(* IEC 61131-3 sources: Std_PalletMover/Class/Wewo_LinkedObjectBase, 1 file *)

(* ---- Wewo_LinkedObjectBase.st ---- *)
(*!
<Class
	Name               = "Wewo_LinkedObjectBase"
	Revision           = "0.10"
	RealtimeTask       = "false"
	CyclicTask         = "false"
	BackgroundTask     = "false"
	Sigmatek           = "false"
	OSInterface        = "false"
	HighPriority       = "false"
	Automatic          = "false"
	UpdateMode         = "Prescan"
	SharedCommandTable = "true"
	Objectsize         = "(654,120)"
	Comment            = "Base class for linked objects&#13;&#10;">
	<Channels>
		<Client Name="p_NextObject" Required="false" Internal="false" Comment="Pointer to next object in linked list"/>
		<Client Name="p_PreviousObject" Required="false" Internal="false" Comment="Pointer to previous object in linked list&#13;&#10;(is automatically filled if p_NextObject is connected)"/>
	</Channels>
	<RevDoku>
		<Owner Company="Safan BV" Author="HenOdi"/>
		<Dokumentation Revision="0.10" Date="2012-03-14" Author="HenOdi" Company="Safan BV" Description="Init() Only set p_NextObject durin initCnt=2&#13;&#10;Prepare to remove methodes (add DO_NOT_USE) in future"/>
		<Dokumentation Revision="0.9" Date="2011-11-22" Author="NieTie" Company="Safan BV" Description="Split up Linked List functionality into&#13;&#10;- Linked List Control base&#13;&#10;- Linked List object base&#13;&#10;&#13;&#10;Remove control functionality from "/>
	</RevDoku>
	<Network Name="Wewo_LinkedObjectBase">
		<!-- List of Components in this network -->
		<Components>
			<Object
				Name       = "_base"
				Class      = "WewoBase"
				Position   = "(218,120)"
				Visualized = "false">
				<Channels>
					<Server Name="m_Id"/>
					<Server Name="m_p_Name"/>
					<Server Name="o_ErrorWarningStatus"/>
					<Server Name="ObjectStatus"/>
					<Server Name="ToObject"/>
					<Client Name="c_Group"/>
					<Client Name="op_LogData"/>
					<Client Name="toOsLibTaskObjControl"/>
				</Channels>
			</Object>
		</Components>
		<Comments>
		</Comments>
		<!-- List of Connections in this network -->
		<Connections>
			<Connection Source="this.ToObject" Destination="_base.ToObject" Vertices="(856,210),(684,210),"/>
			<Connection Source="this.ObjectStatus" Destination="_base.ObjectStatus" Vertices="(856,270),(684,270),"/>
			<Connection Source="this.o_ErrorWarningStatus" Destination="_base.o_ErrorWarningStatus" Vertices="(856,330),(684,330),"/>
			<Connection Source="this.m_Id" Destination="_base.m_Id" Vertices="(856,390),(684,390),"/>
			<Connection Source="this.m_p_Name" Destination="_base.m_p_Name" Vertices="(856,450),(684,450),"/>
			<Connection Source="_base.op_LogData" Destination="this.op_LogData" Vertices="(218,210),(38,210),"/>
			<Connection Source="_base.c_Group" Destination="this.c_Group" Vertices="(218,270),(38,270),"/>
		</Connections>
		<!-- Headerfiles -->
		<Options>
		</Options>
	</Network>
</Class>
*)
#pragma using WewoBase

Wewo_LinkedObjectBase : CLASS
: WewoBase
  //Servers:
  //Clients:
	p_PreviousObject 	: CltChCmd_Wewo_LinkedObjectBase;
	p_NextObject 	: CltChCmd_Wewo_LinkedObjectBase;
  //Variables:
  //Functions:

	FUNCTION VIRTUAL GLOBAL Init;
				//! <Function Comment="Get pointer to previous object in chain list" Name="GetPreviousObjectPtr"/>
	FUNCTION GLOBAL GetPreviousObjectPtr
		VAR_OUTPUT
			p_Object 	: pVoid;
		END_VAR;
				//! <Function Comment="Set pointer to previous object in chain list" Name="SetPreviousObjectPtr"/>
	FUNCTION GLOBAL SetPreviousObjectPtr
		VAR_INPUT
			p_Object 	: pVoid;
		END_VAR;
				//! <Function Comment="Get pointer to next object in chain list" Name="GetNextObjectPtr"/>
	FUNCTION GLOBAL GetNextObjectPtr
		VAR_OUTPUT
			p_Object 	: pVoid;
		END_VAR;
				//! <Function Comment="Set pointer to next object in chain list" Name="SetNextObjectPtr"/>
	FUNCTION GLOBAL SetNextObjectPtr
		VAR_INPUT
			p_Object 	: pVoid;
		END_VAR;
				//! <Function Comment="This methode is reserved for application specific &#13;&#10;functionality that should be handled in a synchronise &#13;&#10;(in sequence of linked list) way." Name="SyncTask"/>
	FUNCTION VIRTUAL GLOBAL SyncTask
		VAR_INPUT
			p_SyncTaskData 	: pVoid;			//! <Variable Comment="Pointer to data(structure) used to handover parameters &#13;&#10;and return data." Name="SyncTask.p_SyncTaskData"/>
		END_VAR
		VAR_OUTPUT
			State 	: BOOL;			//! <Variable Comment="State&#13;&#10;TRUE if OK&#13;&#10;FALSE if failure detected" Name="SyncTask.State"/>
		END_VAR;

	FUNCTION VIRTUAL GLOBAL LinkedListAddObject
		VAR_INPUT
			p_PrevObj 	: pVoid;
		END_VAR
		VAR_OUTPUT
			State 	: DINT;
		END_VAR;

	FUNCTION VIRTUAL GLOBAL LinkedListRemoveObject
		VAR_OUTPUT
			State 	: DINT;
		END_VAR;

	FUNCTION GLOBAL DO_NOT_USE_SearchObjectNextTree
		VAR_INPUT
			ObjectId 	: UDINT;
		END_VAR
		VAR_OUTPUT
			p_Object 	: pVoid;
		END_VAR;

	FUNCTION GLOBAL DO_NOT_USE_SearchObjecPreviousTree
		VAR_INPUT
			ObjectId 	: UDINT;
		END_VAR
		VAR_OUTPUT
			p_Object 	: pVoid;
		END_VAR;
  //Tables:
	FUNCTION @STD
		VAR_OUTPUT
			ret_code	: CONFSTATES;
		END_VAR;
	FUNCTION GLOBAL TAB @CT_;
END_CLASS;

FUNCTION VIRTUAL GLOBAL Wewo_LinkedObjectBase::Init

  WewoBase::Init();
  if initCnt = 2 then
    p_NextObject := p_NextObject.Read();
    if p_NextObject <> NIL then
      p_NextObject^$Wewo_LinkedObjectBase.SetPreviousObjectPtr(p_Object:=this);
    end_if;

  end_if;

END_FUNCTION

(***************************************************************
Wewo_LinkedObjectBase::GetPreviousObjectPtr

Description:    Get pointer to previous object in chain list

Parameter:      -
Return:         Pointer to previous object in chain.
                NIL is returned if no object is connected.
***************************************************************)
FUNCTION GLOBAL Wewo_LinkedObjectBase::GetPreviousObjectPtr
	VAR_OUTPUT
		p_Object 	: pVoid;
	END_VAR

  p_Object := p_PreviousObject;

END_FUNCTION

(***************************************************************
Wewo_LinkedObjectBase::SetPreviousObjectPtr

Description:    Set pointer to previous object in chain list

Parameter:      Pointer to previous object in chain.
Return:         -
***************************************************************)
FUNCTION GLOBAL Wewo_LinkedObjectBase::SetPreviousObjectPtr
	VAR_INPUT
		p_Object 	: pVoid;
	END_VAR

  p_PreviousObject := p_Object;

END_FUNCTION

(***************************************************************
Wewo_LinkedObjectBase::GetNextObjectPtr

Description:    Get pointer to next object in chain list

Parameter:      -
Return:         Pointer to next object in chain.
                NIL is returned if no object is connected.
***************************************************************)
FUNCTION GLOBAL Wewo_LinkedObjectBase::GetNextObjectPtr
	VAR_OUTPUT
		p_Object 	: pVoid;
	END_VAR

  p_Object := p_NextObject;

END_FUNCTION

(***************************************************************
Wewo_LinkedObjectBase::SetNextObjectPtr

Description:    Set pointer to next object in chain list

Parameter:      Pointer to next object in chain.
Return:         -
***************************************************************)
FUNCTION GLOBAL Wewo_LinkedObjectBase::SetNextObjectPtr
	VAR_INPUT
		p_Object 	: pVoid;
	END_VAR

  p_NextObject := p_Object;

END_FUNCTION

#pragma warning (disable : 73)

(***************************************************************
Wewo_LinkedObjectBase::SyncTask

Description:       This methode is reserved for application specific
                   functionality that should be handled in a synchronise
                   (in sequence of linked list) way.

Parameter:         Pointer to data(structure) used to handover parameters
                   and return data.

Return:            State
                   TRUE if OK
                   FALSE if failure detected
***************************************************************)

FUNCTION VIRTUAL GLOBAL Wewo_LinkedObjectBase::SyncTask
	VAR_INPUT
		p_SyncTaskData 	: pVoid;
	END_VAR
	VAR_OUTPUT
		State 	: BOOL;
	END_VAR

  State := FALSE;        // Default return failure, No functionality implemented yet

END_FUNCTION

#pragma warning (default : 73)

//******************************************************************************
// ******************************************************************************
//  START NIET MEER GEBRUIKEN WORDT VERIJDERD
// ********************************************************************************
//******************************************************************************

//***************************************************************
//Wewo_LinkedObjectBase::LinkedListAddObject
//
//Description:       Add object in linked list.
//
//                   situation before this method is called
//                   PrevObj -> (P,2,N)
//                   (P,this,N)
//                   linked list -> (P,1,N)<->(P,2,N)<->(P,3,N)<->NIL
//
//                   situation after this method
//                   linked list -> (P,1,N)<->(P,2,N)<->(P,this,N)<->(P,3,N)->NIL
//
//Parameter:         Pointer to previous object in linked list.
//
//Return:            0  if OK
//                   -1 if SW error
//Note:              This methode is only valid if list is not empty.
//                   First object in list should be set outsite this method.
//***************************************************************
// *******************************************************************************
//  NIET MEER GEBRUIKEN WORDT VERIJDERD
// ********************************************************************************

FUNCTION VIRTUAL GLOBAL Wewo_LinkedObjectBase::LinkedListAddObject
	VAR_INPUT
		p_PrevObj 	: pVoid;
	END_VAR
	VAR_OUTPUT
		State 	: DINT;
	END_VAR

  if p_PrevObj <> NIL then
    // Valid parameter

    // Set Our next and previous pointers
    p_NextObject      := p_PrevObj^$Wewo_LinkedObjectBase.GetNextObjectPtr();
    p_PreviousObject  := p_PrevObj;

    // Set next pointer in previous object
    p_PrevObj^$Wewo_LinkedObjectBase.SetNextObjectPtr(this);

    // Set Previous pointer in next object
    if p_NextObject <> NIL then
      // We are not last object in list
      p_NextObject^$Wewo_LinkedObjectBase.SetPreviousObjectPtr(this);
    end_if;

    State := 0;
  else
  // Error pointer parameter is NIL
    WriteActiveErrorWarning(IntErrorWarningId:= MSGID_NIL_POINTER,
                            LogLevel         := LL_ERROR_INTERNAL,
                            p_msg            := "Wewo_LinkedObjectBase::LinkedListAddObject Error p_PrevObj = NIL"
                           );
    State := -1;

  end_if;

END_FUNCTION

//***************************************************************
//Wewo_LinkedObjectBase::LinkedListRemoveObject
//
//Description:       Remove object from linked list.
//
//                   situation before this method is called
//                   linked list -> (P,1,N)<->(P,this,N)<->(P,3,N)<->NIL
//
//                   situation after this method
//
//                   NIL <-(P,this,N) -> NIL
//                   linked list -> (P,1,N)<->(P,3,N)->NIL
//
//Parameter:         -
//Return:            0  if OK
//                   -1 if SW error
//Note:              0
//***************************************************************
//*******************************************************************************
//  NIET MEER GEBRUIKEN WORDT VERIJDERD
// ********************************************************************************

FUNCTION VIRTUAL GLOBAL Wewo_LinkedObjectBase::LinkedListRemoveObject
	VAR_OUTPUT
		State 	: DINT;
	END_VAR

  // Set previous pointer in next object
  if p_NextObject <> NIL then
    p_NextObject^$Wewo_LinkedObjectBase.SetPreviousObjectPtr(p_Object:=p_PreviousObject);

  end_if;

  // Set next pointer in previous object
  if p_PreviousObject <> NIL then
    p_PreviousObject^$Wewo_LinkedObjectBase.SetNextObjectPtr(p_Object:=p_NextObject);

  end_if;

  // Clear our next and previous pointers
  p_NextObject      := NIL;
  p_PreviousObject  := NIL;

  State := 0;

END_FUNCTION

//***************************************************************
//Wewo_LinkedObjectBase::SearchObjectNextTree
//
//Description:       Searches an  object in linked list via Next pointer.
//                   Object should have an Id filled in m_id.
//
//Parameter:         Object Id.
//
//Return:            pointer to object if found
//                   NIL if not found
//***************************************************************
//*******************************************************************************
//  NIET MEER GEBRUIKEN WORDT VERIJDERD
//********************************************************************************

FUNCTION GLOBAL Wewo_LinkedObjectBase::DO_NOT_USE_SearchObjectNextTree
	VAR_INPUT
		ObjectId 	: UDINT;
	END_VAR
	VAR_OUTPUT
		p_Object 	: pVoid;
	END_VAR

	VAR
    Id       : UDINT;
  END_VAR

  p_Object := this;           // Start searching with this object

  while p_Object <> NIL do
    // Next object available in chain .

    Id := p_Object^$Wewo_LinkedObjectBase.m_Id.Read();

    if ObjectId = Id then
      // Object found,
      exit;             // exit loop

    end_if;

    // Get next object in linked list
    p_Object := p_Object^$Wewo_LinkedObjectBase.GetNextObjectPtr();

  end_while;

END_FUNCTION

// *******************************************************************************
//  NIET MEER GEBRUIKEN WORDT VERIJDERD
// ********************************************************************************

FUNCTION GLOBAL Wewo_LinkedObjectBase::DO_NOT_USE_SearchObjecPreviousTree
	VAR_INPUT
		ObjectId 	: UDINT;
	END_VAR
	VAR_OUTPUT
		p_Object 	: pVoid;
	END_VAR

	VAR
    Id       : UDINT;
  END_VAR

  p_Object := this;           // Start searching with this object

  while p_Object <> NIL do
    // Next object available in chain .

    Id := p_Object^$Wewo_LinkedObjectBase.m_Id.Read();

    if ObjectId = Id then
      // Object found,
      exit;             // exit loop

    end_if;

    // Get previous object in linked list
    p_Object := p_Object^$Wewo_LinkedObjectBase.GetPreviousObjectPtr();

  end_while;

END_FUNCTION

// ******************************************************************************
// *******************************************************************************
//   EIND NIET MEER GEBRUIKEN WORDT VERIJDERD
// *******************************************************************************
// ******************************************************************************
